(* CODESYS project TSR Applikation.project

Project tree, tasks and I/O mapping:
  XV100 : XV400, Eaton Automation, version 3.5.6.0
    application Application
      libraries: SysFile23, * (System); TSR Libary, 1.3 (Eaton Automation); Standard, 3.5.5.0 (System)
      task Task (cyclic, interval t#10ms, priority 1) calls MAIN
      program MAIN [ST]: A0_Start, A1_Einlesen, A2_Prozess, A30_HEADER, A31_PROGRAMM, A300_PROG_NAME, A301_DATE, A302_USER_NAME, A303_LOOP, A310_GOTO, A311_MOV, A312_WAIT, A313_PENUP, A314_PENDOWN, A315_STARTPOINT, A316_CLICK, A317_DOUBLE_CLICK, A3_Befehl_Selection, A4_ComOpen, A5_TSR_Steuern, A50_Pfeiltasten, A61_Syntax, A60_Prozess, A610_HEADER, A611_PROGRAMM, A6_Syntax_Testen, A7_ComClose, B100_Abbruch, B101_AbbruchSTProgramm, B102_AbbruchDirekteSteuerung
      Symbols
      data type wState
*)

// XV100/Application/wState
TYPE wState: 
(
(*0*)	Alles_Ok,
(*1*)	Error_beim_oeffnen,
(*2*)	Error_beim_Senden_von_einem_STRING_durch_das_COM_Port,
(*3*)	Error_beim_Empfangen_von_einem_STRING_durch_das_COM_Port,
(*4*)	Timeout_beim_COM_Port_oeffnen,
(*5*)	Timeout_beim_COM_Port_senden,
(*6*)	Timeout_beim_COM_Port_empfangen,
(*7*)	Es_ist_keine_Verbindunge_mit_dem_TSR_vorhanden,
(*8*)	TSR_hat_keine_korrekte_Antowrt_zurueckgegeben,
(*9*)	Der_TSR_befindet_sich_out_of_range,
(*10*)	Im_Header_des_ST_hat_es_einen_Fehler,
(*11*)	Im_Programm_des_ST_hat_es_einen_Fehler,
(*12*)	Syntax_Fehler_im_ST,
(*13*)	COM_Port_ist_nicht_Geoeffnet,
(*14*)	Timeout_beim_Click_weahrend_dem_Go_to_FB,
(*15*)	Timeout_beim_Click_weahrend_dem_Pen_FB,
(*16*)	Timeout_beim_Connect_weahrend_dem_TSR_COM,
(*17*)  Timeout_beim_Double_Click_weahrend_dem_Go_to_FB,
(*18*)  Timeout_beim_Double_Click_weahrend_dem_Pen_FB,
(*19*)  Timeout_beim_Get_position_weahrend_dem_TSR_COM,
(*20*)	Timeout_beim_Go_to_FB_Weahrend_dem_TSR_COM,
(*21*)	Timeout_beim_Progress_Wait_FB_Weahrend_dem_TSR_COM,
(*22*)	Timeout_beim_Pen_FB_Weahrend_dem_TSR_COM,
(*23*)	Error_beim_schliessen_vom_Com_Port,
(*24*)	Timeout_beim_Com_Port_schliessen
)WORD; 
END_TYPE

// XV100/Application/MAIN
PROGRAM MAIN
VAR
//GUI EIN/AUSGàNGE	
	LTx_StartEinlesen			:BOOL;						//Das Startbool für das einlesen.
	LTx_DoneEinlesen			:BOOL;						//Wird gesetzt wenn das Einlesen vom .txt File zu ende ist.
	LTx_ResetEinlesen			:BOOL;						//Mit diesem Bool löscht man das eingelesen File.
	LTst_DateipfadEinlesen		:STRING := '0';				//Dateipfad bei einlesen.
	LTx_Error					:BOOL;						//Das Error Flag.
	LTst_Array					:ARRAY [0..2000] OF STRING;	//Der Zwischenspeicher vom STRING Array.
	LTst_Line					:STRING;					//Ein Zwischenspeicher der ganzen Linie.
	LTi_ComPort					:INT := 1;					//Der ComPort den man haben will.
	LTx_Connectet				:BOOL;						//Ist die Applikation mit dem TSR verbunden.
	LTx_Abbruch					:BOOL;						//Der Vorgang Abbrechen.
	LTx_HeaderRead				:BOOL;						//Den Header einlesen.
	LTx_ProgrammRead			:BOOL;						//Das Programm einlesen.
	LTst_Dateipfad				:STRING := '\StorageCard\';	//Der Dateipfad String.
	LTx_ProgramON				:BOOL;						//Wenn die Programm Befehle gerade aktiv sind.
	LTx_HeaderDone				:BOOL;						//Wenn der Header eingelesen wurde.
	LTw_wState					:WORD;						//Das Wstate für die HMI
	LTx_SyntaxTest				:BOOL := 1;					//Ist eins wenn die Syntax geteste werden soll.
	LTx_SyntaxOk				:BOOL;						//Ist eins wenn die Syntax ok ist.
	LTi_CounterDurchlauf		:INT;						//Er zählt die Anzahl der durchläufe.
	LTx_ProgrammStop			:BOOL;						//Mit diesem Bool kann man das Programm Stoppen.
	LTx_AbbruchSTProgramm		:BOOL;						//Mit diesem Boll kann man den ST Ausführen vorgang resten.
	LTx_AbbruchDirekteSteuerung	:BOOL;						//Mit diesem Boll bricht man die direkt Steuerung ab.
	LTi_Startpunktx				:INT;						//Der erste Startpunkt
	LTi_Startpunkty				:INT;						//Der zweite Startpunk	
//GUI Die vom Steuerprogramm kommen
	LTst_PROG_NAME				:STRING;					//Wird vom Steuerfile geholt
	LTst_USER_NAME				:STRING;					//""
	LTst_DATE					:STRING;					//""
	LTx_Loop					:BOOL;						//Gibt an ob der Loop verwendet wird.
	
//GUI Die bei Startpoint Teachen benötigt wird.
	LTi_yTeach					:INT;						//Die y Koordinate die getacht werden soll.
	LTi_xTeach					:INT;						//Die x Koordinate die getacht werden soll.
	LTx_GotoTeach				:BOOL;						//Gehe mit den Koordinaten.
	LTx_StartpointTeach			:BOOL;						//Teache diese Koordinate als Startpunkt.
	LTx_TeachenEin				:BOOL;						//Schaltet den Teach Modus ein.

//GUI Variabeln für die Pfeiltasten
	LTi_Step					:INT;						//Die Schritgrösse wie die MOV Befehle sind.
	LTx_PfeilOben				:BOOL;						//Der Pfeil nach oben.
	LTx_PfeilUnten				:BOOL;						//Der Pfeil nach unten.
	LTx_PfeilLinks				:BOOL;						//Der Pfeil nach Links.
	LTx_PfeilRechts				:BOOL;						//Dir Pfeiltasten nach Rechts.
	LTi_xPos					:INT;						//Soll die momentane relavitve Position vom TSR angeben.
	LTi_yPos					:INT;						//Dasselbe wie oben.
	LTx_Unbedinbar				:BOOL;						//Die Pfeiltasten werden dadurch unbdinbar.
	LTx_UnbedinbarPfeilOben		:BOOL;						//Die Pfeiltasten unbedinbar.
	LTx_UnbedinbarPfeilUnten	:BOOL;						//Die Pfeiltasten unbedinbar.
	LTx_UnbedinbarPfeilLinks	:BOOL;						//Die Pfeiltasten unbedienbar Links
	LTx_UnbedinbarPfeilRechts	:BOOL;						//Die Peiltasten ist nicht bedinbar wenn rechts.
	LTx_PenUpTaste				:BOOL;						//Der Pfeil nach oben Taste.
	LTx_PenDownTaste			:BOOL;						//Der Pfeil nach unten Taste.
	LTx_UnbedinbarPenUp			:BOOL;						//Der Pfeil nach oben unbedinbar machen.
	LTx_UnbedinbarPenDown		:BOOL;						//Der Pfeil nach unten unbedinbar machen.
	
//INTERNE VARIABELN
	LTi_ZustandMain				:INT;						//Der Zustand des Main Cases.
	LTi_ZustandEinlesen			:INT;						//Der Zustand des Einlesen Cases.
	LTi_ZustandProzess			:INT;						//Der Zustand des Prozess Cases.
	wState						:wState;					//Der Status für die ENUM Tabelle.
	LTx_TestOn					:BOOL;						//Wenn die Programm Befehle gerade aktiv sind.
	LTi_SyntaxPosx				:INT;						//Die X Position im Syntax test.
	LTi_SyntaxPosy				:INT;						//Die Y Position im Syntax test.
	LTi_maxSyntaxPosx			:INT;						//Die X Position im Syntax test.
	LTi_maxSyntaxPosy			:INT;						//Die Y Position im Syntax test.
					
	//Variabeln für das File Einlesen	
		LTst_DateipfadIntern	:STRING;					//Der Interne Dateipfad.
		LTst_Modus				:STRING;					//Der File Modus wie die Files geöffnet werden.
		LTdw_Handle				:DWORD;						//Der Handle vom Steuerprogramm.
		LTi_ZeichenPos			:INT;						//Die momentane Linie.
		LTst_Temp				:STRING;					//Der Temponäre String.
		LTptby_Temp				:POINTER TO BYTE;			//Der Pointer der auf den STRING zeigt.
		LTptby_Temp1			:POINTER TO BYTE; 			//Der 2. Pointer um eine Linenverschiebung zu ermöglichen.
		LTby_Temp				:BYTE;						//Ein Speicher für das Zeichen.
		LTi_ArrayPosEinlesen	:INT;						//Die ARRAY Position.
		LTi_EndePos				:INT;						//Soll die Position vom Ende einer Zeiler angeben.
	//Variabeln für den Prozess
		LTst_Befehl				:STRING;					//Zwischenspeicher für den Befehl.
		LTi_ArrayPosBefehl		:INT;						//Die Array Position für die Befehle.
		LTst_Information		:STRING;					//Hier werden die Informationen für den Befehl gespeichert.
		LTx_FirstTime			:BOOL;						//Wenn das Programm zu erstem mal hier ist.
		LTi_ArraySize			:INT;						//Die Array Grösse vom File.
		LTx_HeaderON			:BOOL;						//Wenn die Header Befehle gerade aktiv sind.
		
//FUKTIONEN / FUNKTIONSBLÖCKE
	LTfb_TSR_Pen_up_down			:TSR_Pen_up_down;
	LTfb_Connect_with_TSR			:Connect_with_TSR;
	LTfb_Move_TSR_xy				:FB_Move_TSR_xy;
	LTfb_Go_to_TSR_xy				:FB_Go_to_TSR_xy;
	LTfb_Timer						:TON;
	LTfb_Click						:FB_Click;
	LTfb_Double_Click				:FB_Double_Click;
	LTfb_Get_TSR_Pos				:FB_Get_TSR_position;	// Get Pos FB
END_VAR

CASE LTi_ZustandMain OF
	0:
		A0_Start();					//Prüfe die Startbedingungen.
	1:
		A1_Einlesen();				//Lese Das SteuerFile ein.
	2:
		A2_Prozess();				//Werte den Befehl des Steuerfiles aus.
	3:
		A3_Befehl_Selection();		//Die Befehle auswählen.
	4:
		A4_ComOpen();				//Mach den ComPort auf.
	5:
		A5_TSR_Steuern();			//Der TSR soll Steuerbar sein.
	6:
		A6_Syntax_Testen();			//Die Syntax des Eingelesenen Programmes Testen.
END_CASE

LTw_wState := wState;
B100_Abbruch();
B101_AbbruchSTProgramm();	
B102_AbbruchDirekteSteuerung();				
//Funktionsblöcke aufrufen
	LTfb_TSR_Pen_up_down();			
	LTfb_Connect_with_TSR();				
	LTfb_Move_TSR_xy();					
	LTfb_Go_to_TSR_xy();
	LTfb_Click();
	LTfb_Double_Click();				
	LTfb_Timer();
	LTfb_Get_TSR_Pos();

ACTION A0_Start:
IF LTx_StartEinlesen THEN							//Wenn eingelesen werden soll.
	LTx_StartEinlesen := 0;							//Boll zurücksetzten.
	LTi_ZustandMain := 1;							//Setzte den Zustand auf 1 um das Einlesen zu starten.
END_IF

IF (LTx_HeaderRead OR LTx_ProgrammRead) AND LTx_DoneEinlesen THEN		//Wenn der Prozess gestartet werden sollte und ein File eingelesn ist.
		LTi_ZustandMain := 2;							//Setzte den Zustand auf 2 um den Prozess zu starten.
		LTi_ArrayPosBefehl := 0;						//Die Array Pos setzten.
END_IF

IF LTx_TeachenEin THEN								//Wenn der startpoint touch boutten ein ist
	LTi_ZustandMain := 5;							//In den Teach modus wechseln.
END_IF
END_ACTION

ACTION A1_Einlesen:
//Den Internen Dateipfad setzen.
LTst_DateipfadIntern := CONCAT(LTst_Dateipfad, CONCAT(LTst_DateipfadEinlesen, '.txt'));

//Das File öffnen
LTst_Modus := 'r';
LTdw_Handle := SysFileOpen(FileName := LTst_DateipfadIntern, Mode := LTst_Modus);

//Linien Lesen. 
//Tu das solange nicht das ende vom File erreicht ist.
WHILE NOT SysFileEOF(LTdw_Handle) DO
	LTst_Temp := '';							//Den Temp speicher Leeren
	LTi_ZeichenPos := 0;						//Linie													
	LTptby_Temp := ADR(LTst_Temp);				//Adresse im Pointer Speichern										

//Solange noch gelesen wird
WHILE (SysFileRead(File:= LTdw_Handle, Buffer:= ADR(LTby_Temp), Size := 1) = 1) DO
//Den Pointer um eine Stelle verschieben
LTptby_Temp1 := LTptby_Temp + LTi_ZeichenPos;													
//Das gelesene Byte im Temp String bei der richtigen Position speichern
LTptby_Temp1^ := LTby_Temp;
//Wenn im Temp ein 0A ist soll der vorgang abrechen
IF LTby_Temp = 16#0A OR (LTi_ZeichenPos >= 80)
THEN																					
	EXIT;
END_IF;	
LTi_ZeichenPos := LTi_ZeichenPos + 1;			//Zähle die Pos höher

END_WHILE
//Speicher die Zeile im Array String
LTi_EndePos := FIND(LTst_Temp,'$R$L');
LTst_Array[LTi_ArrayPosEinlesen] := LEFT(STR := LTst_Temp, SIZE := LTi_EndePos - 1);
LTi_ArrayPosEinlesen := LTi_ArrayPosEinlesen + 1;
END_WHILE

SysFileClose(File:= LTdw_Handle);

IF LTx_SyntaxTest THEN
	LTi_ZustandMain := 6;
	LTi_xPos := 0;
	LTi_yPos := 0;
ELSE
	LTi_ZustandMain := 0;
END_IF

LTi_ArrayPosEinlesen := 0;
LTx_HeaderDone := 0;
LTx_DoneEinlesen := 1;
END_ACTION

ACTION A2_Prozess:
IF LTx_ProgrammRead OR LTx_HeaderRead THEN						//Wenn das Programm angehalten wird 
	IF LTx_ProgrammStop THEN
		LTx_ProgrammRead := 0;
		LTx_ProgrammStop := 0;
	ELSE
	IF 0 < FIND(LTst_Array[LTi_ArrayPosBefehl], '//') THEN
		LTst_Line := LEFT(LTst_Array[LTi_ArrayPosBefehl], Size := FIND(LTst_Array[LTi_ArrayPosBefehl], '//') - 1);	//Kommentar vom rest trennen.
	ELSE
		LTst_Line := LTst_Array[LTi_ArrayPosBefehl];
	END_IF
	IF NOT (LTst_Line = '') THEN						//wenn im rest immernoch etwas drin ist dann.
		WHILE FIND(LTst_Line, ' ') > 0 DO				//Lösche alle Leerzeichen
			LTst_Line := DELETE(LTst_Line, 1, FIND(LTst_Line, ' ')); 
		END_WHILE
		WHILE FIND(LTst_Line, '$t') > 0 DO				//und Lösche alle tabulatoren, Das ist nicht nötig da die tabulatoren beim einlesen Gelöscht werden.
			LTst_Line := DELETE(LTst_Line, 1, FIND(LTst_Line, '$t')); 
		END_WHILE
		IF NOT (LTst_Line = '') THEN					//Ist jetzt noch etwas im STRING?
														//Ist schon eine Verbindung zum TSR aufgebaut.
			IF LTx_Connectet = 0 THEN
				LTi_ZustandMain := 4;
			ELSE
				LTi_ZustandMain := 3;
			END_IF										//Wenn ja gehe
		END_IF	
	END_IF																	
//Zur Position vom nächsten Befehl gehen.
LTi_ArrayPosBefehl := LTi_ArrayPosBefehl +1;
	END_IF
END_IF
END_ACTION

ACTION A30_HEADER:
//Hier werden alle HEADER Informationen übertragen
//Der Programm Name	
IF 0 < FIND(LTst_Line, 		'PROG_NAME=') 		THEN
	A300_PROG_NAME();

//Das Datum
ELSIF 0 < FIND(LTst_Line,	'DATE=')				THEN
	A301_DATE();

//übernimmt das Datum
ELSIF 0 < FIND(LTst_Line, 	'USER_NAME=') 		THEN
	A302_USER_NAME();

//Führt den Loop befehl aus
ELSIF 0 < FIND(LTst_Line, 	'LOOP=') 				THEN
	A303_LOOP();

//Ansonsten Error ausgeben
ELSE 
	LTx_Error := 1;
	wState	:= 10;				//Error in Header	
	LTi_ZustandMain := 0;
END_IF
END_ACTION

ACTION A31_PROGRAMM:
//Diese Befehle dürfen nur im Programm sein
//GO TO Befehl
IF 0 < FIND(LTst_Line, 			'GOTO')			THEN
	A310_GOTO();

//MOV Befehl
ELSIF 0 < FIND(LTst_Line, 		'MOV')			THEN
	A311_MOV();

//Das Warten
ELSIF 0 < FIND(LTst_Line, 		'WAIT')			THEN
	A312_WAIT();

//Pen up
ELSIF 0 < FIND(LTst_Line, 		'PENUP')		THEN
	A313_PENUP();

//Pen down
ELSIF 0 < FIND(LTst_Line, 		'PENDOWN') 		THEN
	A314_PENDOWN();

//startpunkt
ELSIF 0 < FIND(LTst_Line, 		'STARTPOINT')	THEN
	A315_STARTPOINT();

//Double click
ELSIF 0 < FIND(LTst_Line, 		'DCLICK')		THEN	//Die frage nach DClick muss vor dem Click sein weil er ansonsten den Click sieht.
	A317_DOUBLE_CLICK();
	
//click	
ELSIF 0 < FIND(LTst_Line, 		'CLICK')		THEN
	A316_CLICK();

//Ansonsten Error ausgeben
ELSE
	LTx_Error := 1;
	wState	:= 11;				//Error in Programm
	LTi_ZustandMain := 0;
END_IF
END_ACTION

ACTION A300_PROG_NAME:
LTst_PROG_NAME := DELETE(LTst_Line, 10, 1);
LTi_ZustandMain := 2;
END_ACTION

ACTION A301_DATE:
LTst_DATE := DELETE(LTst_Line, 5, 1);
LTi_ZustandMain := 2;
END_ACTION

ACTION A302_USER_NAME:
LTst_USER_NAME := DELETE(LTst_Line, 10, 1);
LTi_ZustandMain := 2;
END_ACTION

ACTION A303_LOOP:
//Wenn das Loop ein ist schalte auf loop um
IF DELETE(LTst_Line, 5, 1) = 'ON' THEN
	LTx_Loop := 1;
ELSE
	LTx_Loop := 0;
END_IF
LTi_ZustandMain := 2;
END_ACTION

ACTION A310_GOTO:
LTst_Information := DELETE(LTst_Line, 4, 1);

LTfb_Go_to_TSR_xy(
	xExecute:= 1, 
	iGotox:=STRING_TO_INT(LEFT(STR:=LTst_Information, Size := FIND(LTst_Information, ':') - 1)) , 
	iGotoy:=STRING_TO_INT(RIGHT(STR:=LTst_Information, Size := LEN(LTst_Information) - FIND(LTst_Information, ':'))),);
	

IF LTfb_Go_to_TSR_xy.xDone THEN
	LTi_ZustandMain := 2;			//Zurück zum letzten Befehl.
	LTfb_Go_to_TSR_xy(				//Sezte den FB zurück.
	xExecute:= 0, );
END_IF

IF LTfb_Go_to_TSR_xy.xError THEN
	LTx_Error := 1;
	wState := LTfb_Go_to_TSR_xy.wState;
END_IF
END_ACTION

ACTION A311_MOV:
LTst_Information := DELETE(LTst_Line, 3, 1);

LTfb_Move_TSR_xy(
	xExecute:=1 , 
	iMovx:=STRING_TO_INT(LEFT(STR:=LTst_Information, Size := FIND(LTst_Information, ':') - 1)) , 
	iMovy:=STRING_TO_INT(RIGHT(STR:=LTst_Information, Size := LEN(LTst_Information) - FIND(LTst_Information, ':'))),);

IF LTfb_Move_TSR_xy.xDone THEN
	LTi_ZustandMain := 2;			//Zurück zum letzten Befehl.
	LTfb_Move_TSR_xy(				//Sezte den FB zurück.
	xExecute:= 0, );
END_IF

IF LTfb_Move_TSR_xy.xError THEN
	LTx_Error := 1;
	wState := LTfb_Move_TSR_xy.wState;
END_IF
END_ACTION

ACTION A312_WAIT:
LTst_Information := DELETE(LTst_Line, 4, 1);

IF LTx_FirstTime = 0 THEN
LTx_FirstTime := 1;
LTfb_Timer(IN := 1, PT:= STRING_TO_TIME(CONCAT('T#',CONCAT(LTst_Information,'ms'))));	//Setzte den Timer.
END_IF


IF LTfb_Timer.Q THEN					//Wenn der Timer Abgelaufen ist.
		LTi_ZustandMain := 2;		//In den Error Zustand gehen.
		LTfb_Timer.IN := 0;
		LTx_FirstTime := 0;
END_IF

LTfb_Timer();
END_ACTION

ACTION A313_PENUP:
LTst_Information := DELETE(LTst_Line, 5, 1);

//Hier Wird der Stift nach oben bewegt.
LTfb_TSR_Pen_up_down(					//FB PEN aufruf.
	xExecute:= 1, 
	xPen:= 0, );

IF LTfb_TSR_Pen_up_down.xDone THEN	//Wenn der FB fertig ist.
	LTi_ZustandMain := 2;			//Zurück zum letzten Befehl.
	LTfb_TSR_Pen_up_down(				//Sezte den FB zurück.
	xExecute:= 0, );
END_IF

IF LTfb_TSR_Pen_up_down.xError THEN
	LTx_Error := 1;
	wState := LTfb_TSR_Pen_up_down.wState;
END_IF
END_ACTION

ACTION A314_PENDOWN:
LTst_Information := DELETE(LTst_Line, 7, 1);


//Hier Wird der Stift nach unten bewegt.
LTfb_TSR_Pen_up_down(					//FB PEN aufruf.
	xExecute:= 1, 
	xPen:= 1, );

IF LTfb_TSR_Pen_up_down.xDone THEN	//Wenn der FB fertig ist.
	LTi_ZustandMain := 2;			//Zurück zum letzten Befehl.
	LTfb_TSR_Pen_up_down(				//Sezte den FB zurück.
	xExecute:= 0, );
END_IF

IF LTfb_TSR_Pen_up_down.xError THEN
	LTx_Error := 1;
	wState := LTfb_TSR_Pen_up_down.wState;
END_IF
END_ACTION

ACTION A315_STARTPOINT:
LTst_Information := DELETE(LTst_Line, 10, 1);

//Lade die werte in die Funktion.
FN_Set_TSR_startpoint(iStartpointx:=STRING_TO_INT(LEFT(STR:=LTst_Information, Size := FIND(LTst_Information, ':') - 1)) , 
iStartpointy:=STRING_TO_INT(RIGHT(STR:=LTst_Information, Size := LEN(LTst_Information) - FIND(LTst_Information, ':'))),);
//Gehe zurück zum selcet
LTi_ZustandMain := 2;
END_ACTION

ACTION A316_CLICK:
LTst_Information := DELETE(LTst_Line, 5, 1);

LTfb_Click
(
	xExecute:= 1, 
	iKlicktox:=STRING_TO_INT(LEFT(STR:=LTst_Information, Size := FIND(LTst_Information, ':') - 1)) , 
	iKlicktoy:=STRING_TO_INT(RIGHT(STR:=LTst_Information, Size := LEN(LTst_Information) - FIND(LTst_Information, ':'))),
);
	

IF LTfb_Click.xDone THEN
	LTi_ZustandMain := 2;			//Zurück zum letzten Befehl.
	LTfb_Click(						//Sezte den FB zurück.
	xExecute:= 0, );
END_IF

IF LTfb_Click.xError THEN
	LTx_Error := 1;
	wState := LTfb_Click.wState;
END_IF
END_ACTION

ACTION A317_DOUBLE_CLICK:
LTst_Information := DELETE(LTst_Line, 7, 1);

LTfb_Double_Click(
	xExecute:= 1, 
	iKlicktox:=STRING_TO_INT(LEFT(STR:=LTst_Information, Size := FIND(LTst_Information, ':') - 1)) , 
	iKlicktoy:=STRING_TO_INT(RIGHT(STR:=LTst_Information, Size := LEN(LTst_Information) - FIND(LTst_Information, ':'))),);
	

IF LTfb_Double_Click.xDone THEN
	LTi_ZustandMain := 2;			//Zurück zum letzten Befehl.
	LTfb_Double_Click(						//Sezte den FB zurück.
	xExecute:= 0, );
END_IF

IF LTfb_Double_Click.xError THEN
	LTx_Error := 1;
	wState := LTfb_Double_Click.wState;
END_IF
END_ACTION

ACTION A3_Befehl_Selection:
//Entscheiden ob es ein Header oder Program befehl ist.
	IF LTx_HeaderRead THEN
	
		//Der Header End
		IF LTst_Line 		= 	'HEADER_END' 		THEN
			LTx_HeaderON := 0;
			LTi_ZustandMain := 0;
			LTx_HeaderRead := 0; 
			LTx_HeaderDone := 1;
		//Wenn der Header eingeschaltete ist
		ELSIF LTx_HeaderON THEN
			A30_HEADER();			//Geh zum Header Befehlsatz
		//Beim Header Start
		ELSIF LTst_Line		= 	'HEADER_START' 		THEN
			LTx_HeaderON := 1;
			LTi_ZustandMain := 2;	//Da das Programm zu Ende ist.
			wState := 0;			//Alles ist Ok
		ELSE
			LTi_ZustandMain := 2;	//Gehe zur nächsten Zeile
		END_IF
	
	ELSIF LTx_ProgrammRead THEN
		
		//Wenn das Programm Endet
		IF LTst_Line 		= 	'PROGRAMM_END' 		THEN
			LTx_ProgramON := 0;
			LTi_ZustandMain := 0;	//Da das Programm zu Ende ist.
			wState := 0;			//Alles ist Ok.
			LTi_CounterDurchlauf := LTi_CounterDurchlauf + 1;
			IF LTx_Loop THEN
				LTx_ProgrammRead := 1;
			ELSE
				LTx_ProgrammRead := 0;
			END_IF
		//Wenn man im Programm ist
		ELSIF LTx_ProgramON THEN
			A31_PROGRAMM();			//Geh zum Programm Befehlsatz
		//Programm Start
		ELSIF LTst_Line 		= 	'PROGRAMM_START' 	THEN
			LTx_ProgramON := 1;
			LTi_ZustandMain :=2;	//Gehe zur nächsten Zeile
		ELSE
			LTi_ZustandMain := 2;	//Gehe zur nächsten Zeile
		END_IF
	//Wenn man Gleichzeitig im Header und im Programm ist gibt Error aus.
	ELSIF LTx_ProgramON AND LTx_HeaderON THEN
		LTx_Error := 0;				//Error setzten
		wState := 12;				//Syntax Fehler
		LTi_ZustandMain := 0;		//Zum Main zurückehren.
	
	ELSE
		LTi_ZustandMain := 2;		//zum nächstem zustand.
	END_IF
END_ACTION

ACTION A4_ComOpen:
LTfb_Connect_with_TSR(
	xExecute:=1 , 
	iCom:=LTi_ComPort, 
	xPort := 1);
	
IF LTfb_Connect_with_TSR.xDone THEN
	LTi_ZustandMain := 3;	//Starte den Prozess
	LTx_Connectet := 1;		//Setzte verbindung
	LTfb_Connect_with_TSR(
	xExecute:=0 ,);
END_IF

IF LTfb_Connect_with_TSR.xError THEN
	LTx_Error := 1;
	wState := LTfb_Connect_with_TSR.wState;
END_IF
END_ACTION

ACTION A5_TSR_Steuern:
//Wenn der Com Port nicht offen ist dann den Comport öffnen
IF LTx_Connectet = 0 THEN
	LTfb_Connect_with_TSR(
	xExecute:=1 , 
	iCom:=LTi_ComPort ,
	xPort := 1,);
	
	IF LTfb_Connect_with_TSR.xDone THEN	//Ist der Com Port offen?
		LTx_Connectet := 1;		//Setzte verbindung
		LTfb_Connect_with_TSR(
		xExecute:=0 ,);
	END_IF
	
	IF LTfb_Connect_with_TSR.xError THEN
		LTx_Connectet := 0;
		LTx_Error := 1;
		wState := LTfb_Connect_with_TSR.wState;
	END_IF
ELSE
	A50_Pfeiltasten();				//Mit den Pfeiltasten den TSR bewegen.
	LTi_ZustandMain := 0;
END_IF
END_ACTION

ACTION A50_Pfeiltasten:
IF LTfb_Get_TSR_Pos.xExecute = 1 THEN
	LTfb_Get_TSR_Pos();
	
	IF LTfb_Get_TSR_Pos.xDone THEN
		LTi_xPos := LTfb_Get_TSR_Pos.iPosx + LTi_Startpunktx;
		LTi_yPos := LTfb_Get_TSR_Pos.iPosy + LTi_Startpunkty;
		LTfb_Get_TSR_Pos(				//Sezte den FB zurück.
		xExecute:= 0,);
	END_IF
	
	IF LTfb_Get_TSR_Pos.xError THEN
		LTx_Error := 1;
		wState := LTfb_Get_TSR_Pos.wState;
	END_IF

ELSIF LTx_PfeilOben THEN			//Wenn die Pfeil taste nach oben gedrückt ist.
	LTfb_Move_TSR_xy(			//aufruf des fb moves.
	xExecute := 1,
	iMovy:= -LTi_Step,);
	LTx_Unbedinbar := 1;

ELSIF LTx_PfeilUnten THEN		//wenn die Pfiel taste nach unten gedrückt ist
	LTfb_Move_TSR_xy(		//Aufruf des FB Moves
	xExecute := 1,
	iMovy:= LTi_Step,);
	LTx_Unbedinbar := 1;

ELSIF LTx_PfeilLinks THEN		//Wen die Pfeil Taste nach links gedrückt ist.
	LTfb_Move_TSR_xy(		//Aufruf des FB Moves
	xExecute := 1,
	iMovx:= -LTi_Step,);
	LTx_Unbedinbar := 1;

ELSIF LTx_PfeilRechts THEN		//Wenn die Pfeil taste nach rechts gedrückt. ist
	LTfb_Move_TSR_xy(		//Aufruf des FB Moves
	xExecute := 1,	
	iMovx:= LTi_Step,);
	LTx_Unbedinbar := 1;

ELSIF LTx_GotoTeach THEN	//Wenn man die GOTO werte teachen will
	LTfb_Go_to_TSR_xy(
	xExecute:= 1, 
	iGotox:=LTi_xTeach,
	iGotoy:=LTi_yTeach,);
	LTx_Unbedinbar := 1;


	
	IF LTfb_Go_to_TSR_xy.xDone THEN
		LTfb_Go_to_TSR_xy(				//Sezte den FB zurück.
		xExecute:= 0, );
		LTx_GotoTeach := 0;
		LTx_Unbedinbar := 0;
	END_IF
		
	IF LTfb_Go_to_TSR_xy.xError THEN
		LTx_Error := 1;
		wState := LTfb_Go_to_TSR_xy.wState;
	END_IF
	
ELSIF LTx_PenUpTaste THEN
	LTfb_TSR_Pen_up_down(
	xExecute := 1,
	xPen := 0,);
	LTx_Unbedinbar := 1;
	
	IF LTfb_TSR_Pen_up_down.xDone THEN
		LTfb_TSR_Pen_up_down(
		xExecute := 0,);
		LTx_Unbedinbar := 0;
		LTx_UnbedinbarPenUp := 1;
		LTx_UnbedinbarPenDown := 0;
		LTx_PenUpTaste := 0;
	END_IF
	
	IF LTfb_TSR_Pen_up_down.xError THEN
		LTx_Error := 1;
		wState := LTfb_TSR_Pen_up_down.wState;
	END_IF

ELSIF LTx_PenDownTaste THEN
	LTfb_TSR_Pen_up_down(
	xExecute := 1,
	xPen := 1,);
	LTx_Unbedinbar := 1;
	
	IF LTfb_TSR_Pen_up_down.xDone THEN
		LTfb_TSR_Pen_up_down(
		xExecute := 0,);
		LTx_Unbedinbar := 0;
		LTx_UnbedinbarPenDown := 1;
		LTx_UnbedinbarPenUp := 0;
		LTx_PenDownTaste := 0;
	END_IF
	
	IF LTfb_TSR_Pen_up_down.xError THEN
		LTx_Error := 1;
		wState := LTfb_TSR_Pen_up_down.wState;
	END_IF
		
ELSIF LTx_StartpointTeach THEN
	//Lade die werte in die Funktion.
	LTx_StartpointTeach := 0;
	LTi_Startpunktx	 := LTi_xPos;
	LTi_Startpunkty  := LTi_yPos;	
	FN_Set_TSR_startpoint(iStartpointx:=LTi_Startpunktx	, iStartpointy:=LTi_Startpunkty	,); 
	IF LTx_SyntaxTest THEN
		IF LTi_maxSyntaxPosx + LTi_Startpunktx	 > 313 OR LTi_maxSyntaxPosy + LTi_Startpunkty	> 226 OR LTi_SyntaxPosy + LTi_Startpunkty < 0 OR LTi_SyntaxPosx + LTi_Startpunktx < 0 THEN
			LTx_Error := 1;
			wState := 9;
			LTi_ZustandMain := 0;
			LTx_SyntaxOk := 0;
		END_IF	
	END_IF
ELSE 
	LTfb_Get_TSR_Pos(
	xExecute:=1 ,);
END_IF	


IF LTfb_Move_TSR_xy.xDone THEN	//Alles zurücksetzten
	LTfb_Move_TSR_xy(
	xExecute:= 0,
	iMovx := 0,
	iMovy := 0,);
	LTx_Unbedinbar := 0;
	LTx_PfeilOben := 0; 
	LTx_PfeilUnten := 0;
	LTx_PfeilLinks := 0;
	LTx_PfeilRechts := 0;
END_IF


//Out of range Prüfen.	
IF LTfb_Move_TSR_xy.xError THEN
	LTx_Error := 1;
	wState := LTfb_Move_TSR_xy.wState;
END_IF

IF LTi_xPos + LTi_Step > 313 THEN
	LTx_UnbedinbarPfeilRechts := 1;
ELSE
	LTx_UnbedinbarPfeilRechts := 0;
END_IF

IF LTi_xPos - LTi_Step < 0 THEN
	LTx_UnbedinbarPfeilLinks := 1;
ELSE
	LTx_UnbedinbarPfeilLinks := 0;
END_IF

IF LTi_yPos + LTi_Step > 226 THEN
	LTx_UnbedinbarPfeilUnten := 1;
ELSE
	LTx_UnbedinbarPfeilUnten := 0;
END_IF

IF LTi_yPos - LTi_Step < 0 THEN
	LTx_UnbedinbarPfeilOben := 1;
ELSE
	LTx_UnbedinbarPfeilOben := 0;
END_IF
END_ACTION

ACTION A61_Syntax:
//Entscheiden ob es ein Header oder Program befehl ist.

	
		//Der Header End
		IF LTst_Line 		= 	'HEADER_END' 		THEN
			LTx_HeaderON := 0;
			LTi_ZustandMain := 6;
			LTx_HeaderRead := 0; 
		//Wenn der Header eingeschaltete ist
		ELSIF LTx_HeaderON THEN
			A610_HEADER();			//Geh zum Header Befehlsatz
		//Beim Header Start
		ELSIF LTst_Line		= 	'HEADER_START' 		THEN
			LTx_HeaderON := 1;
			LTi_ZustandMain := 6;	//Da das Programm zu Ende ist.
			wState := 0;			//Alles ist Ok
		ELSE
			LTi_ZustandMain := 6;	//Gehe zur nächsten Zeile
		END_IF
	

		
		//Wenn das Programm Endet
		IF LTst_Line 		= 	'PROGRAMM_END' 		THEN
			LTx_TestON := 0;
			LTi_ZustandMain := 0;	//Da das Programm zu Ende ist.
			wState := 0;			//Alles ist Ok
			LTx_HeaderRead := 1;
			LTx_StartpointTeach := 0;
		//Wenn man im Programm ist
		ELSIF LTx_TestON THEN
			A611_PROGRAMM();			//Geh zum Programm Befehlsatz
		//Programm Start
		ELSIF LTst_Line 		= 	'PROGRAMM_START' 	THEN
			LTx_TestOn := 1;
			LTi_ZustandMain := 6;	//Gehe zur nächsten Zeile
		ELSE
			LTi_ZustandMain := 6;	//Gehe zur nächsten Zeile
		END_IF
	//Wenn man Gleichzeitig im Header und im Programm ist gibt Error aus.
	IF LTx_TestON AND LTx_HeaderON THEN
		LTx_Error := 1;				//Error setzten
		wState := 12;				//Syntax Fehler
		LTi_ZustandMain := 0;		//Zum Main zurückehren.
	END_IF
END_ACTION

ACTION A60_Prozess:
//In diesem Prozess werden die Befhele im Eingelesenem String so vorbereitet das Das man mit dem
//String einen Syntax Test machen kann. Dieser Prozess ist sehr ähnlich wie der Prozess von A1_Einlesen.

	
IF 0 < FIND(LTst_Array[LTi_ArrayPosBefehl], '//') THEN
		LTst_Line := LEFT(LTst_Array[LTi_ArrayPosBefehl], Size := FIND(LTst_Array[LTi_ArrayPosBefehl], '//') - 1);	//Kommentar vom rest trennen.
ELSE
		LTst_Line := LTst_Array[LTi_ArrayPosBefehl];
END_IF
IF NOT (LTst_Line = '') THEN						//wenn im rest immernoch etwas drin ist dann.
	WHILE FIND(LTst_Line, ' ') > 0 DO				//Lösche alle Leerzeichen
		LTst_Line := DELETE(LTst_Line, 1, FIND(LTst_Line, ' ')); 
	END_WHILE
	WHILE FIND(LTst_Line, '$t') > 0 DO				//und Lösche alle tabulatoren, Das ist nicht nötig da die tabulatoren beim einlesen Gelöscht werden.
		LTst_Line := DELETE(LTst_Line, 1, FIND(LTst_Line, '$t')); 
	END_WHILE
	IF NOT (LTst_Line = '') THEN					//Ist jetzt noch etwas im STRING?
		LTi_ZustandMain	:= 0; 						//Der Main Zustand.
	END_IF
END_IF
													//Rufe die Syntax Prüfung auf
LTi_ArrayPosBefehl := LTi_ArrayPosBefehl +1;		//Zähle die Position Hoch
END_ACTION

ACTION A610_HEADER:
//Hier werden alle HEADER Informationen übertragen
//Der Programm Name	
IF 0 < FIND(LTst_Line, 		'PROG_NAME=') 		THEN
	LTx_SyntaxOk := 1;
//Das Datum
ELSIF 0 < FIND(LTst_Line,	'DATE=')			THEN
	LTx_SyntaxOk := 1;
//übernimmt das Datum
ELSIF 0 < FIND(LTst_Line, 	'USER_NAME=') 		THEN
	LTx_SyntaxOk := 1;
//Führt den Loop befehl aus
ELSIF 0 < FIND(LTst_Line, 	'LOOP=') 			THEN
	LTx_SyntaxOk := 1;
//Ansonsten Error ausgeben
ELSE 
	LTx_Error := 1;
	wState	:= 10;				//Error in Header	
	LTi_ZustandMain := 0;
	Ltx_SyntaxOk := 0;
END_IF
END_ACTION

ACTION A611_PROGRAMM:
//Diese Befehle dürfen nur im Programm sein
//GO TO Befehl
IF 0 < FIND(LTst_Line, 			'GOTO')			THEN
	LTx_SyntaxOk := 1;
	LTst_Information := DELETE(LTst_Line, 4, 1);
	LTi_SyntaxPosx := STRING_TO_INT(LEFT(STR:=LTst_Information, Size := FIND(LTst_Information, ':') - 1));
	LTi_SyntaxPosy := STRING_TO_INT(RIGHT(STR:=LTst_Information, Size := LEN(LTst_Information) - FIND(LTst_Information, ':')));


	
//MOV Befehl
ELSIF 0 < FIND(LTst_Line, 		'MOV')			THEN
	LTx_SyntaxOk := 1;
	LTst_Information := DELETE(LTst_Line, 3, 1);
	LTi_SyntaxPosx := LTi_SyntaxPosx + STRING_TO_INT(LEFT(STR:=LTst_Information, Size := FIND(LTst_Information, ':') - 1));
	LTi_SyntaxPosy := LTi_SyntaxPosy + STRING_TO_INT(RIGHT(STR:=LTst_Information, Size := LEN(LTst_Information) - FIND(LTst_Information, ':')));

//Das Warten
ELSIF 0 < FIND(LTst_Line, 		'WAIT')			THEN
	LTx_SyntaxOk := 1;

//Pen up
ELSIF 0 < FIND(LTst_Line, 		'PENUP')		THEN
	LTx_SyntaxOk := 1;

//Pen down
ELSIF 0 < FIND(LTst_Line, 		'PENDOWN') 		THEN
	LTx_SyntaxOk := 1;

//startpunkt
ELSIF 0 < FIND(LTst_Line, 		'STARTPOINT')	THEN
	LTx_SyntaxOk := 1;
	LTi_Startpunktx :=STRING_TO_INT(LEFT(STR:=LTst_Information, Size := FIND(LTst_Information, ':') - 1));
	LTi_Startpunkty :=STRING_TO_INT(RIGHT(STR:=LTst_Information, Size := LEN(LTst_Information) - FIND(LTst_Information, ':')));

//Double click
ELSIF 0 < FIND(LTst_Line, 		'DCLICK')		THEN	//Die frage nach DClick muss vor dem Click sein weil er ansonsten den Click sieht.
	LTx_SyntaxOk := 1;
	LTst_Information := DELETE(LTst_Line, 6, 1);
	LTi_SyntaxPosx := STRING_TO_INT(LEFT(STR:=LTst_Information, Size := FIND(LTst_Information, ':') - 1));
	LTi_SyntaxPosy := STRING_TO_INT(RIGHT(STR:=LTst_Information, Size := LEN(LTst_Information) - FIND(LTst_Information, ':')));

//click	
ELSIF 0 < FIND(LTst_Line, 		'CLICK')		THEN
	LTx_SyntaxOk := 1;
	LTst_Information := DELETE(LTst_Line, 5, 1);
	LTi_SyntaxPosx := STRING_TO_INT(LEFT(STR:=LTst_Information, Size := FIND(LTst_Information, ':') - 1));
	LTi_SyntaxPosy := STRING_TO_INT(RIGHT(STR:=LTst_Information, Size := LEN(LTst_Information) - FIND(LTst_Information, ':')));

//Ansonsten Error ausgeben
ELSE
	LTx_Error := 1;
	wState	:= 11;				//Error in Programm
	LTi_ZustandMain := 0;
	Ltx_SyntaxOk := 0;
END_IF

IF LTi_SyntaxPosx > LTi_maxSyntaxPosx THEN
	LTi_maxSyntaxPosx := LTi_SyntaxPosx;
END_IF

IF LTi_SyntaxPosy > LTi_maxSyntaxPosy THEN
	LTi_maxSyntaxPosy := LTi_SyntaxPosy;
END_IF

IF LTi_SyntaxPosx + LTi_Startpunktx	 > 313 OR LTi_SyntaxPosy + LTi_Startpunkty	> 226 OR LTi_SyntaxPosy + LTi_Startpunkty < 0 OR LTi_SyntaxPosx + LTi_Startpunktx < 0 THEN
	LTx_Error := 1;
	wState := 9;
	LTi_ZustandMain := 0;
	LTx_SyntaxOk := 0;
END_IF
END_ACTION

ACTION A6_Syntax_Testen:
IF LTx_SyntaxTest THEN
	A60_Prozess();
	A61_Syntax();
END_IF
END_ACTION

ACTION A7_ComClose:
LTfb_Connect_with_TSR(
	xExecute:=1 , 
	iCom:=LTi_ComPort, 
	xPort := 0);
	
IF LTfb_Connect_with_TSR.xDone THEN
	LTx_Connectet := 0;		//Setzte verbindung
	LTfb_Connect_with_TSR(
	xExecute:=0 ,);
END_IF

IF LTfb_Connect_with_TSR.xError THEN
	LTx_Error := 1;
	wState := LTfb_Connect_with_TSR.wState;
END_IF
END_ACTION

ACTION B100_Abbruch:
IF LTx_Abbruch THEN
	LTi_ZustandMain := 0;		//Zum urzustand zurück
	LTx_HeaderON := 0;
	Ltx_ProgramOn := 0;
	LTx_HeaderRead := 0; 
	LTx_ProgrammRead := 0;
	LTi_ArrayPosBefehl := 0;
	LTx_HeaderDone := 0;
	LTx_DoneEinlesen := 0;
	LTx_FirstTime := 0;
	LTx_SyntaxOk := 0;
	LTi_SyntaxPosx := 0;
	LTi_SyntaxPosy := 0;
	LTi_CounterDurchlauf := 0;
	
	//GUI Informationen zurücksetzten
	LTst_PROG_NAME			:= '';					
	LTst_USER_NAME			:= '';					
	LTst_DATE				:= '';					
	LTx_Loop				:= 0;					

	//Teach Funktion zurücketzten
	LTx_Connectet := 0;
	LTx_GotoTeach := 0;
	LTx_StartpointTeach := 0;
	LTx_Unbedinbar := 0;
	
	//Die Funktionsblöcke zurücksezten
	LTfb_TSR_Pen_up_down.xExecute := 0;			
	LTfb_Connect_with_TSR.xExecute := 0;				
	LTfb_Move_TSR_xy.xExecute := 0;					
	LTfb_Go_to_TSR_xy.xExecute := 0;
	LTfb_Click.xExecute := 0;
	LTfb_Double_Click.xExecute := 0;
	LTfb_Get_TSR_Pos.xExecute := 0;				
	LTfb_Timer.IN := 0;	

	//Die Errors zurücksetzten
	LTx_Error := 0;
	wState := 0;
	LTx_PfeilOben := 0; 
	LTx_PfeilUnten := 0;
	LTx_PfeilLinks := 0;
	LTx_PfeilRechts := 0;
	LTi_Step := 0;		

	//FB's aufrufen um zurückzusetzten
	LTfb_TSR_Pen_up_down();			
	LTfb_Connect_with_TSR();				
	LTfb_Move_TSR_xy();					
	LTfb_Go_to_TSR_xy();
	LTfb_Click();
	LTfb_Double_Click();				
	LTfb_Timer();
	LTfb_Get_TSR_Pos();	
		
	IF LTx_Connectet THEN
		A7_ComClose();
	ELSE
		LTx_Abbruch := 0;
	END_IF
END_IF
END_ACTION

ACTION B101_AbbruchSTProgramm:
IF LTx_AbbruchSTProgramm THEN
	LTx_AbbruchSTProgramm := 0;
	LTi_ZustandMain := 0;		//Zum urzustand zurück
	Ltx_ProgramOn := 0;
	LTx_ProgrammRead := 0;
	LTi_CounterDurchlauf := 0;
		
	//Die Funktionsblöcke zurücksezten
	LTfb_TSR_Pen_up_down.xExecute := 0;			
	LTfb_Connect_with_TSR.xExecute := 0;				
	LTfb_Move_TSR_xy.xExecute := 0;					
	LTfb_Go_to_TSR_xy.xExecute := 0;
	LTfb_Click.xExecute := 0;
	LTfb_Double_Click.xExecute := 0;
	LTfb_Get_TSR_Pos.xExecute := 0;				
	LTfb_Timer.IN := 0;	
	LTx_FirstTime := 0;
	//Die Errors zurücksetzten
	LTx_Error := 0;
	wState := 0;
END_IF
END_ACTION

ACTION B102_AbbruchDirekteSteuerung:
IF LTx_AbbruchDirekteSteuerung THEN
	LTx_Unbedinbar := 1;
	LTi_ZustandMain := 0;		//Zum urzustand zurück
	LTx_FirstTime := 0;
	
	//Teach Funktion zurücketzten
	LTx_GotoTeach := 0;
	LTx_StartpointTeach := 0;
	LTx_TeachenEin := 0;
	LTi_Startpunktx	:= 0;
	LTi_Startpunkty	:= 0;
	FN_Set_TSR_startpoint(iStartpointx:=0	, iStartpointy:=0	,); 

	
	//Die Funktionsblöcke zurücksezten
	LTfb_TSR_Pen_up_down.xExecute := 0;						
	LTfb_Move_TSR_xy.xExecute := 0;					
	LTfb_Go_to_TSR_xy.xExecute := 0;
	LTfb_Click.xExecute := 0;
	LTfb_Double_Click.xExecute := 0;
	LTfb_Get_TSR_Pos.xExecute := 0;				
	LTfb_Timer.IN := 0;	

	//Die Errors zurücksetzten
	LTx_Error := 0;
	wState := 0;
	LTx_PfeilOben := 0; 
	LTx_PfeilUnten := 0;
	LTx_PfeilLinks := 0;
	LTx_PfeilRechts := 0;
	LTi_Step := 0;		

	//FB's aufrufen um zurückzusetzten
	LTfb_TSR_Pen_up_down();			
	LTfb_Connect_with_TSR();				
	LTfb_Move_TSR_xy();					
	LTfb_Go_to_TSR_xy();
	LTfb_Click();
	LTfb_Double_Click();				
	LTfb_Timer();
	LTfb_Get_TSR_Pos();			

	LTx_AbbruchDirekteSteuerung := 0;
	LTx_TeachenEin := 1;
	LTx_Unbedinbar := 0;

END_IF
END_ACTION

END_PROGRAM
